(* CoDeSys 2.3 export: GlobalVariableList.ftl *)

(* Global variable list: ${name} *)
VAR_GLOBAL<#if constant!false> CONSTANT</#if>

<#if vars?has_content>
<#list vars as var>
    ${var.name}: ${var.type}<#if var.value??> := ${var.value}</#if>;
</#list>
</#if>

END_VAR
